PROGRAM MAIN
VAR
	_Count			: UINT;
END_VAR

_Count := _Count + 1;

END_PROGRAM

(* stored: Version 1.1.0.1
   POU MAIN: Id {1dbd0600-e9db-4819-b291-3e96fdb29dcc}, SpecialFunc None *)
